SUBAPPLICATION AX_TON_MERGE_QXA_OPC (* 1 Kanal einer geschalteten Gruppe (z.B. Scheinwerfer): nimmt den Toggle-Zustand eines gemeinsamen TOGGLE_RPC_MASTER_QXA_OPC ueber den MASTER-Socket entgegen, verzoegert das Einschalten um PT (AX_TON, Ausschalten sofort), verknuepft per AX_OR_2 mit dem bestehenden IO-Test-Kommando dieses Kanals und treibt den physischen Ausgang. Fuer einen komplett eigenstaendigen Kanal (eigener SoftKey, kein gemeinsamer Master) stattdessen TOGGLE_RPC_MERGE_QXA_OPC oder MERGE_SWITCH_1_QXA_OPC verwenden. *)
  (* Standard: 61499-2; Description: Copyright (c) 2026 Meisterschulen am Ostbahnhof This program and the accompanying materials are made available under the terms of the Eclipse Public License 2.0 which is available at https://www.eclipse.org/legal/epl-2.0/ SPDX-License-Identifier: EPL-2.0 *)
  (* Version 1.0, 2026-09-07, Franz Höpfinger, Meisterschulen am Ostbahnhof, initial API and implementation and/or initial documentation - Scheinwerfer-Kanal, versetztes Einschalten (PT je Instanz unterschiedlich) gegen kapazitive Einschaltstrom-Spitzen *)
  PACKAGE MyLib::sys;
  IMPORT logiBUS::io::DQ::logiBUS_DO;
  IMPORT logiBUS::io::DQ::logiBUS_DO_S;
  (* Documentation:
  1 Kanal einer Klick-Toggle-Gruppe, zeitversetzt hochfahrend
   Nimmt ueber den MASTER-Socket den gemeinsamen Toggle-Zustand eines TOGGLE_RPC_MASTER_QXA_OPC entgegen (mehrere Kanaele koennen sich denselben Master teilen - gemeinsam per AdapterConnections im selben SubApp-Netzwerk verdrahtet, kein OPC-UA noetig). AX_TON verzoegert nur das EINSCHALTEN um PT (je Kanal unterschiedlich, z.B. 0/800/1600ms...) - Ausschalten erfolgt sofort. Danach wie gewohnt per AX_OR_2 mit dem bestehenden IO-Test-Kommando dieses Kanals zusammengefuehrt.
   Praxisbeispiel: Scheinwerfer-Bank mit 6 LED-Kanaelen, EIN SoftKey (ueber TOGGLE_RPC_MASTER_QXA_OPC), aber 6 AX_TON_MERGE_QXA_OPC-Instanzen mit gestaffeltem PT - verteilt den Einschaltstrom der LED-Treiber ueber die Zeit statt alle kapazitiven Lasten gleichzeitig zu schalten.
  *)
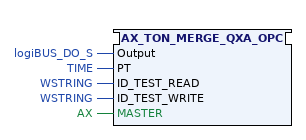
  VAR_INPUT
    Output : logiBUS::io::DQ::logiBUS_DO_S := logiBUS_DO::Invalid; (* Physischer Ausgang dieses Kanals *)
    PT : TIME := T#0ms; (* Einschaltverzoegerung dieses Kanals gegenueber dem Master-Toggle (je Instanz unterschiedlich setzen, z.B. T#0ms/T#800ms/T#1600ms/...) - Ausschalten ist immer sofort *)
    ID_TEST_READ : WSTRING; (* Bestehende IO-Test-Subscribe-Adresse dieses Kanals (z.B. STG5_Q0x_READ) *)
    ID_TEST_WRITE : WSTRING; (* Bestehende IO-Test-Publish-Adresse dieses Kanals (z.B. STG5_Q0x_WRITE) - EIGENER Knoten, NICHT ID_TEST_READs Knoten (sonst Selbstrueckkopplung/Latch, siehe OPC_UA_VERNETZUNG.md Punkt 10+11) *)
  END_VAR
  SOCKETS
    MASTER : adapter::types::unidirectional::AX; (* Toggle-Zustand vom gemeinsamen TOGGLE_RPC_MASTER_QXA_OPC.OUT *)
  END_SOCKETS
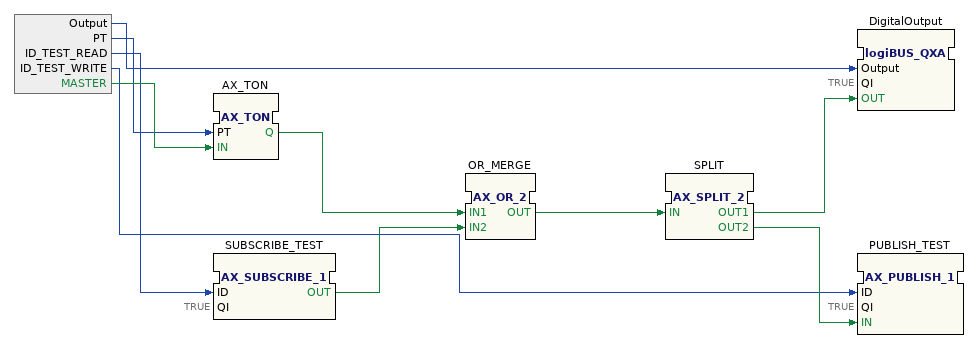
  FBS
    AX_TON : adapter::events::unidirectional::timers::AX_TON;
    SUBSCRIBE_TEST : adapter::net::AX_SUBSCRIBE_1(QI := TRUE);
    OR_MERGE : adapter::booleanOperators::AX_OR_2;
    DigitalOutput : logiBUS::io::DQ::logiBUS_QXA(QI := TRUE);
    SPLIT : adapter::events::unidirectional::AX_SPLIT_2;
    PUBLISH_TEST : adapter::net::AX_PUBLISH_1(QI := TRUE);
  END_FBS
  DATA_CONNECTIONS
    Output TO DigitalOutput.Output;
    PT TO AX_TON.PT;
    ID_TEST_READ TO SUBSCRIBE_TEST.ID;
    ID_TEST_WRITE TO PUBLISH_TEST.ID;
  END_CONNECTIONS
  ADAPTER_CONNECTIONS
    MASTER TO AX_TON.IN;
    AX_TON.Q TO OR_MERGE.IN1;
    SUBSCRIBE_TEST.OUT TO OR_MERGE.IN2;
    OR_MERGE.OUT TO SPLIT.IN;
    SPLIT.OUT1 TO DigitalOutput.OUT;
    SPLIT.OUT2 TO PUBLISH_TEST.IN;
  END_CONNECTIONS
END_SUBAPPLICATION
